FUNCTION CompareAnyType : BOOL
VAR_INPUT
	a					: __SYSTEM.AnyType; // a and b have to be same type
	is					: ComparisonOperator;
	b					: __SYSTEM.AnyType; // a and b have to be same type
END_VAR

CASE is OF
	ComparisonOperator.Equal:
		CompareAnyType := IsEqualAnyType(a, b);
	ComparisonOperator.NotEqual:
		CompareAnyType := IsNotEqualAnyType(a, b);
	ComparisonOperator.LessThan:
		CompareAnyType := IsLessThanAnyType(a, b);
	ComparisonOperator.LessThanOrEqual:
		CompareAnyType := IsLessThanOrEqualAnyType(a, b);
	ComparisonOperator.GreaterThan:
		CompareAnyType := IsGreaterThanAnyType(a, b);
	ComparisonOperator.GreaterThanOrEqual:
		CompareAnyType := IsGreaterThanOrEqualAnyType(a, b);
END_CASE

END_FUNCTION

(* stored: Version 1.1.0.1
   POU CompareAnyType: Id {dc8e7778-ffdf-0c00-303f-c009e7cd2375}, SpecialFunc None *)
